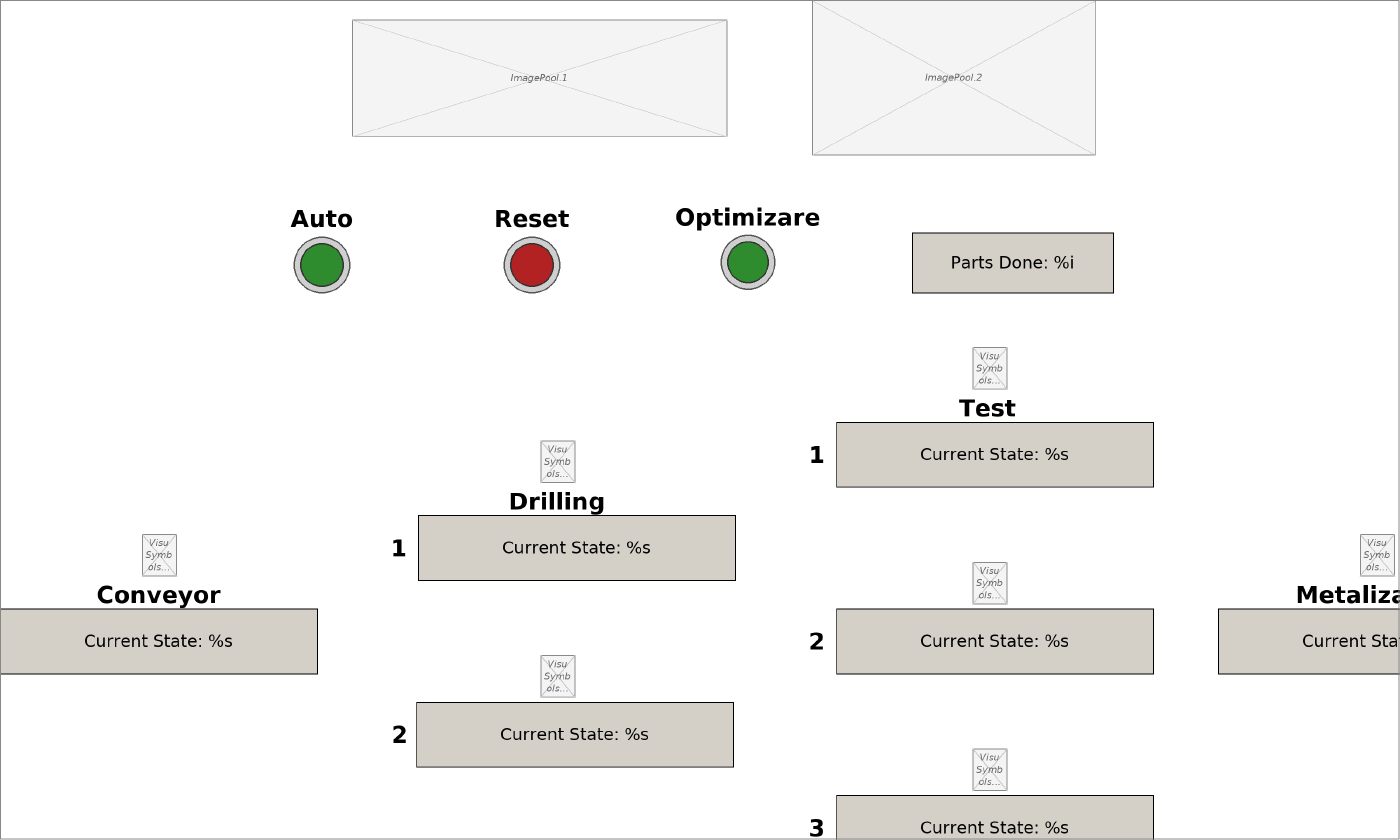
VISUALIZATION Visualization  // 1500x900
    Group (0,0 1500x900)
        Group (377,0 708x162)
            Image (1,75 16x16)
            Image (0,21 402x125), image: ImagePool.1
            Image (493,0 304x166), image: ImagePool.2
        Group (270,218 923x98)
            RoundedRectangle (707,31 216x65), "Parts Done: %i", text variable: Global_Vars.NoOfPartsDone
            Group (0,1 133x97)
                Lamp1 (35,30 80x70), variable: PRG_Cell.m_StartAuto, style: Lamp-Lamp1-Green
                Label (0,0 150x30), "Auto"
            Group (225,1 133x97)
                Lamp1 (35,30 80x70), variable: PRG_Cell.m_ResetRobot, style: Lamp-Lamp1-Red
                Label (0,0 150x30), "Reset"
            Group (450,0 163x97)
                Lamp1 (46,29 71x68), variable: PRG_Cell.Instance_Robot.m_OptOn, style: Lamp-Lamp1-Green
                Label (0,0 163x29), "Optimizare"
        Group (0,372 1462x535)
            Group (0,200 340x150)
                Group (0,50 340x100)
                    RoundedRectangle (0,30 340x70), "Current State: %s", text variable: PRG_Cell.Instance_Conveyor.SFCCurrentStep, colour toggle: PRG_Cell.Instance_Conveyor.m_PartExists
                    Label (95,0 150x30), "Conveyor"
                Image (152,0 37x45), invisible if: not PRG_Cell.Instance_Robot.Position[0], image: VisuSymbols.Symbols.ArrowBoldDown
            Group (407,100 381x350)
                Label (115,50 150x30), "Drilling"
                Group (0,80 381x70)
                    RoundedRectangle (41,0 340x70), "Current State: %s", text variable: PRG_Cell.Instance_Drilling1.SFCCurrentStep, colour toggle: PRG_Cell.Instance_Drilling1.o_PartExists
                    Label (0,20 41x30), "1"
                RoundedRectangle (39,280 340x70), "Current State: %s", text variable: PRG_Cell.Instance_Drilling.SFCCurrentStep, colour toggle: PRG_Cell.Instance_Drilling.o_PartExists
                Label (1,300 41x30), "2"
                Image (172,0 37x45), invisible if: not PRG_Cell.Instance_Robot.Position[1], image: VisuSymbols.Symbols.ArrowBoldDown
                Image (172,230 37x45), invisible if: not PRG_Cell.Instance_Robot.Position[2], image: VisuSymbols.Symbols.ArrowBoldDown
            Group (855,0 381x550)
                Group (0,50 381x100)
                    Label (128,0 150x30), "Test"
                    Group (0,30 381x70)
                        RoundedRectangle (41,0 340x70), "Current State: %s", text variable: PRG_Cell.Instance_Test_1.SFCCurrentStep, colour toggle: PRG_Cell.Instance_Test_1.o_PartExists
                            OnMouseClick: OpenDialog OpenModal=True, OpenCentered=True
                        Label (0,20 41x30), "1"
                Group (0,280 381x70)
                    RoundedRectangle (41,0 340x70), "Current State: %s", text variable: PRG_Cell.Instance_Test_2.SFCCurrentStep, colour toggle: PRG_Cell.Instance_Test_2.o_PartExists
                    Label (0,20 41x30), "2"
                Group (0,480 381x70)
                    RoundedRectangle (41,0 340x70), "Current State: %s", text variable: PRG_Cell.Instance_Test_3.SFCCurrentStep, colour toggle: PRG_Cell.Instance_Test_3.o_PartExists
                    Label (0,20 41x30), "3"
                Image (187,0 37x45), invisible if: not PRG_Cell.Instance_Robot.Position[3], image: VisuSymbols.Symbols.ArrowBoldDown
                Image (187,230 37x45), invisible if: not PRG_Cell.Instance_Robot.Position[4], image: VisuSymbols.Symbols.ArrowBoldDown
                Image (187,430 37x45), invisible if: not PRG_Cell.Instance_Robot.Position[5], image: VisuSymbols.Symbols.ArrowBoldDown
            Group (1305,200 340x150)
                RoundedRectangle (0,80 340x70), "Current State: %s", text variable: PRG_Cell.Instance_Metalization.SFCCurrentStep, colour toggle: PRG_Cell.Instance_Metalization
                Label (74,50 193x30), "Metalization"
                Image (152,0 37x45), invisible if: Not PRG_Cell.Instance_Robot.Position[6], image: VisuSymbols.Symbols.ArrowBoldDown
END_VISUALIZATION

(* stored: Version 1.1.0.1, ProductVersion 3.1.4024.3
   Visu Visualization: Id {59084b05-d032-42ae-a309-0ee92386aa15} *)
